  [993] = {x=-5.4E-05, y=-145.676355, z=-9E-06, rx=0.299285, ry=175.773671, rz=18.534843, fatherId=world[0]}
  [994] = {x=-5.4E-05, y=-145.823252, z=-9E-06, rx=0.299284, ry=175.773671, rz=18.534844, fatherId=world[0]}
  [995] = {x=-5.4E-05, y=-145.970149, z=-9E-06, rx=0.299283, ry=175.773671, rz=18.534845, fatherId=world[0]}
  [996] = {x=-5.4E-05, y=-146.117047, z=-9E-06, rx=0.299282, ry=175.773672, rz=18.534846, fatherId=world[0]}
  [997] = {x=-5.4E-05, y=-146.263944, z=-1E-05, rx=0.299281, ry=175.773672, rz=18.534847, fatherId=world[0]}
  [998] = {x=-5.4E-05, y=-146.410841, z=-1E-05, rx=0.29928, ry=175.773672, rz=18.534848, fatherId=world[0]}
  [999] = {x=-5.4E-05, y=-146.557738, z=-1E-05, rx=0.299279, ry=175.773672, rz=18.534849, fatherId=world[0]}
public mdesc mNomSpeed
